PROGRAM PRG_LVCP2_PowerMeasurement
VAR
	// Enerji Yönetimi
	fbEL3453	: FB_EL3453;	
	stEL3453	: stEL3453;
END_VAR


	fbEL3453(pOut := ADR(stEL3453));

END_PROGRAM

(* stored: Version 1.1.0.1, ProductVersion 3.1.4024.15
   POU PRG_LVCP2_PowerMeasurement: Id {7e5628c9-edef-4634-8dff-23dd194ebd67}, SpecialFunc None *)
